PROGRAM MAIN
VAR
END_VAR

END_PROGRAM

(* stored: Version 1.1.0.1
   POU MAIN: Id {f277e443-3cfc-4f4e-a5fe-9f10589c7ad1} *)
